(* IEC 61131-3 sources: beckhoffAutomationInterface/ST/Shark/Lib/Math, 6 files *)

(* ---- F_IsWithinAbsoluteTolerance.st ---- *)
(* Checks if the measured value is within an absolute tolerance of the setpoint. *)
FUNCTION F_IsWithinAbsoluteTolerance : BOOL
VAR_INPUT
    rMeasured           : LREAL;            // Current measured value
    rSetpoint           : LREAL;            // Target setpoint
    rToleranceAbsolute  : LREAL;            // Tolerance in engineering units (e.g., 0.5)
    bEnabled            : BOOL := FALSE;    // Active flag
END_VAR
VAR
    rError : LREAL;
END_VAR

    // Not at setpoint if disabled
    IF NOT bEnabled THEN
        F_IsWithinAbsoluteTolerance := FALSE;
        RETURN;
    END_IF

    // Calculate absolute error and check against tolerance
    rError := ABS(rMeasured - rSetpoint);
    F_IsWithinAbsoluteTolerance := rError <= rToleranceAbsolute;

END_FUNCTION

(* ---- F_IsWithinTolerance.st ---- *)
(* Checks if measured value is within percentage tolerance of setpoint. *)
FUNCTION F_IsWithinTolerance : BOOL
VAR_INPUT
    rMeasured          : LREAL;    // Current measured value
    rSetpoint          : LREAL;    // Target setpoint
    rTolerancePercent  : LREAL;    // Tolerance as percentage (e.g., 2.0 = 2%)
    bEnabled           : BOOL;     // Controller must be enabled
END_VAR
VAR
    rTolerance : LREAL;
    rError     : LREAL;
END_VAR

    // Not at setpoint if disabled or zero setpoint
    IF NOT bEnabled OR rSetpoint = 0.0 THEN
        F_IsWithinTolerance := FALSE;
        RETURN;
    END_IF

    // Calculate tolerance band and check
    rTolerance := ABS(rSetpoint * rTolerancePercent / 100.0);
    rError := ABS(rMeasured - rSetpoint);
    F_IsWithinTolerance := rError <= rTolerance;

END_FUNCTION

(* ---- F_ModAbs.st ---- *)
(* Positive modulo — returns a value in [0, rModulus).
   Standard MOD can return negative results for negative inputs;
   this function wraps into the positive range. *)
FUNCTION F_ModAbs : LREAL
VAR_INPUT
    rValue   : LREAL;
    rModulus : LREAL;
END_VAR
VAR
    rResult : LREAL;
END_VAR
    IF rModulus = 0.0 THEN
        F_ModAbs := 0.0;
        RETURN;
    END_IF

    rResult := rValue - FLOOR(rValue / rModulus) * rModulus;
    F_ModAbs := rResult;
END_FUNCTION

(* ---- F_RampRateToVelocity.st ---- *)
(* Converts ramp rate from °C/min to velocity °C/sec. *)
FUNCTION F_RampRateToVelocity : LREAL
VAR_INPUT
    rRate_DegPerMin : LREAL;  // Ramp rate in degrees per minute
END_VAR
VAR CONSTANT
    SECONDS_PER_MINUTE : LREAL := 60.0;
END_VAR
    F_RampRateToVelocity := rRate_DegPerMin / SECONDS_PER_MINUTE;
END_FUNCTION

(* ---- F_ScaleRealToInt.st ---- *)
(*
Scales a REAL physics value into an INT raw count format for memory overriding.
Used heavily in the Simulation PRG to spoof Beckhoff A/D terminal behavior.

Formula: Output = (Input - InMin) / (InMax - InMin) * (OutMax - OutMin) + OutMin

Rules observed: Functional Preference (Pure generic math).
*)
FUNCTION F_ScaleRealToInt : INT
VAR_INPUT
    rValue   : REAL;  // The calculated physics engine value (e.g., 150.5 °C)
    rInMin   : REAL;  // The physical minimum (e.g., 0.0 °C)
    rInMax   : REAL;  // The physical maximum (e.g., 300.0 °C)
    nOutMin  : INT;   // The analog minimum (e.g., 0)
    nOutMax  : INT;   // The analog maximum (e.g., 32767)
END_VAR
VAR
    rPercent : REAL;
    rOutTemp : REAL;
END_VAR

// Fail-fast / Division by zero protection
IF (rInMax - rInMin) = 0.0 THEN
    F_ScaleRealToInt := nOutMin;
    RETURN;
END_IF

// Calculate purely
rPercent := (rValue - rInMin) / (rInMax - rInMin);
rOutTemp := (rPercent * INT_TO_REAL(nOutMax - nOutMin)) + INT_TO_REAL(nOutMin);

// Clipping to prevent overflow wrap-around in memory
IF rOutTemp > 32767.0 THEN
    F_ScaleRealToInt := 32767;
ELSIF rOutTemp < -32768.0 THEN
    F_ScaleRealToInt := -32768;
ELSE
    F_ScaleRealToInt := REAL_TO_INT(rOutTemp);
END_IF

END_FUNCTION

(* ---- F_VelocityToRampRate.st ---- *)
(* Converts velocity from °C/sec to ramp rate °C/min. *)
FUNCTION F_VelocityToRampRate : LREAL
VAR_INPUT
    rVelocity_DegPerSec : LREAL;  // Velocity in degrees per second
END_VAR
VAR CONSTANT
    SECONDS_PER_MINUTE : LREAL := 60.0;
END_VAR
    F_VelocityToRampRate := rVelocity_DegPerSec * SECONDS_PER_MINUTE;
END_FUNCTION
